FUNCTION TFOVEMClearAllCommand : bool
VAR_INPUT
Command : POINTER TO Ovem_Command;
END_VAR
VAR
END_VAR

Command^.ErrorReset := FALSE;
Command^.Aspirazione_OFF:=FALSE;
Command^.Aspirazione_ON :=FALSE;
Command^.Aspirazione_ON_ScritturaSoglia:=FALSE;
Command^.ErrorReset := FALSE;
Command^.ErrorReset := FALSE;
Command^.ScriviParametri:= FALSE;

TFOVEMClearAllCommand:=TRUE;

END_FUNCTION

(* stored: Version 1.1.0.1, ProductVersion 3.1.4024.11
   POU TFOVEMClearAllCommand: Id {8d289c92-c297-4847-ba3e-b8d459ee70da}, SpecialFunc None *)
